// TIA Portal V17 export
// export: Created 2024-09-03T21:54:49.3245379Z, ExportSetting WithDefaults, DisplayName Totally Integrated Automation Portal, DisplayVersion V17 Update 7, DisplayName TIA Portal Openness, DisplayVersion V17 Update 7, DisplayName TIA Portal Version Control Interface, DisplayVersion V17, DisplayName SINAMICS Startdrive Advanced, DisplayVersion V17 SP2, DisplayName SINAMICS Startdrive G110M, G120, G120C, G120D, G120P, G115D, DisplayVersion V17 SP2, DisplayName SINAMICS Startdrive G130, G150, S120, S150, SINAMICS MV, S210, DisplayVersion V17 SP2, DisplayName STEP 7 Professional, DisplayVersion V17 Update 7, DisplayName STEP 7 Safety, DisplayVersion V17 Update 6, DisplayName WinCC Advanced / Unified PC, DisplayVersion V17 Update 7
DATA_BLOCK "HydraulicMain_DB"   // DB55
VERSION : 0.1
// stored: AutoNumber true, DBAccessibleFromOPCUA true, DBAccessibleFromWebserver true, InstanceOfName HydraulicMain, InstanceOfType FB
"HydraulicMain"
   // VAR
   //    HydraulicCylinder_LeftCupforming { S7_SetPoint := 'True'} : "HydraulicCylinder";
   //    HydraulicCylinder_RightCupforming { S7_SetPoint := 'True'} : "HydraulicCylinder";
   //    VH1StatusOld { S7_SetPoint := 'True'} : "UDT_Cylinder";
   //    VH2StatusOld { S7_SetPoint := 'True'} : "UDT_Cylinder";
   //    VH3StatusOld { S7_SetPoint := 'True'} : "UDT_Cylinder";
   //    VH4StatusOld { S7_SetPoint := 'True'} : "UDT_Cylinder";
   //    FittingCycle_InstanceCupformingLeft { S7_SetPoint := 'True'} : "FittingCycle";
   //    FittingCycle_InstanceCupformingRight { S7_SetPoint := 'True'} : "FittingCycle";
   //    R_TRIG_Instance { S7_SetPoint := 'True'} : R_TRIG;
   //    R_TRIG_Instance_1 { S7_SetPoint := 'True'} : R_TRIG;
   //    R_TRIG_Instance_2 { S7_SetPoint := 'True'} : R_TRIG;
   //    R_TRIG_Instance_3 { S7_SetPoint := 'True'} : R_TRIG;
   //    HydraulicMotor_Instance { S7_SetPoint := 'True'} : "HydraulicMotor";
   //    dummyCylinderLeft { ExternalAccessible := 'False'; ExternalVisible := 'False'; ExternalWritable := 'False'} : "UDT_Cylinder";
   //    dummyCylinderRight { S7_SetPoint := 'True'} : "UDT_Cylinder";
   // END_VAR
BEGIN
   HydraulicCylinder_LeftCupforming.HydraulicActive := FALSE;
   HydraulicCylinder_LeftCupforming.BasicPositionMin := -5.0;
   HydraulicCylinder_LeftCupforming.BasicPositionMax := 10.0;
   HydraulicCylinder_LeftCupforming.MaxPosition := 105.0;
   HydraulicCylinder_LeftCupforming.ManualCommand := 0;
   HydraulicCylinder_LeftCupforming.CylinderNumber := 3;
   HydraulicCylinder_LeftCupforming.dataOld.Pressure := 0.0;
   HydraulicCylinder_LeftCupforming.dataOld.Flow := 0.0;
   HydraulicCylinder_LeftCupforming.dataOld.Position := 0.0;
   HydraulicCylinder_LeftCupforming.dataOld.StandstillPosition := 0.0;
   HydraulicCylinder_LeftCupforming.dataOld.PressureCmd := 0.0;
   HydraulicCylinder_LeftCupforming.dataOld.FlowCmd := 0.0;
   HydraulicCylinder_LeftCupforming.dataOld.PressureBack := 0.0;
   HydraulicCylinder_LeftCupforming.dataOld.FlowBack := 0.0;
   HydraulicCylinder_LeftCupforming.dataOld.HAxis := 0.0;
   HydraulicCylinder_LeftCupforming.dataOld.Force := 0.0;
   HydraulicCylinder_LeftCupforming.dataOld.Status.InWp := FALSE;
   HydraulicCylinder_LeftCupforming.dataOld.Status.InBp := TRUE;
   HydraulicCylinder_LeftCupforming.dataOld.Status.InFp := TRUE;
   HydraulicCylinder_LeftCupforming.dataOld.Status.ToWp := FALSE;
   HydraulicCylinder_LeftCupforming.dataOld.Status.ToBp := FALSE;
   HydraulicCylinder_LeftCupforming.dataOld.Status.ToFp := TRUE;
   HydraulicCylinder_LeftCupforming.noCollision := TRUE;
   HydraulicCylinder_LeftCupforming.IEC_Timer_0_Instance.PT := T#3S;
   HydraulicCylinder_LeftCupforming.IEC_Timer_0_Instance.IN := FALSE;
   HydraulicCylinder_LeftCupforming.R_TRIG_Instance.CLK := TRUE;
   HydraulicCylinder_LeftCupforming.R_TRIG_Instance.Q := FALSE;
   HydraulicCylinder_LeftCupforming.R_TRIG_Instance.Stat_Bit := TRUE;
   HydraulicCylinder_LeftCupforming.difference := -0.01085043;
   HydraulicCylinder_LeftCupforming.re := -0.1085043;
   HydraulicCylinder_LeftCupforming.IEC_Timer_0_Instance_1.PT := T#400MS;
   HydraulicCylinder_LeftCupforming.IEC_Timer_0_Instance_1.IN := TRUE;
   HydraulicCylinder_LeftCupforming.RampFunction_Instance.Output := 0.0;
   HydraulicCylinder_LeftCupforming.RampFunction_Instance.ErrorBits := 16#0000_0000;
   HydraulicCylinder_RightCupforming.HydraulicActive := FALSE;
   HydraulicCylinder_RightCupforming.BasicPositionMin := -5.0;
   HydraulicCylinder_RightCupforming.BasicPositionMax := 10.0;
   HydraulicCylinder_RightCupforming.MaxPosition := 105.0;
   HydraulicCylinder_RightCupforming.ManualCommand := 0;
   HydraulicCylinder_RightCupforming.CylinderNumber := 4;
   HydraulicCylinder_RightCupforming.dataOld.Pressure := 0.0;
   HydraulicCylinder_RightCupforming.dataOld.Flow := 0.0;
   HydraulicCylinder_RightCupforming.dataOld.Position := 0.0;
   HydraulicCylinder_RightCupforming.dataOld.StandstillPosition := 0.0;
   HydraulicCylinder_RightCupforming.dataOld.PressureCmd := 0.0;
   HydraulicCylinder_RightCupforming.dataOld.FlowCmd := 0.0;
   HydraulicCylinder_RightCupforming.dataOld.PressureBack := 0.0;
   HydraulicCylinder_RightCupforming.dataOld.FlowBack := 0.0;
   HydraulicCylinder_RightCupforming.dataOld.HAxis := 0.0;
   HydraulicCylinder_RightCupforming.dataOld.Force := 0.0;
   HydraulicCylinder_RightCupforming.dataOld.Status.InWp := FALSE;
   HydraulicCylinder_RightCupforming.dataOld.Status.InBp := TRUE;
   HydraulicCylinder_RightCupforming.dataOld.Status.InFp := TRUE;
   HydraulicCylinder_RightCupforming.dataOld.Status.ToWp := FALSE;
   HydraulicCylinder_RightCupforming.dataOld.Status.ToBp := FALSE;
   HydraulicCylinder_RightCupforming.dataOld.Status.ToFp := TRUE;
   HydraulicCylinder_RightCupforming.noCollision := TRUE;
   HydraulicCylinder_RightCupforming.IEC_Timer_0_Instance.PT := T#3S;
   HydraulicCylinder_RightCupforming.IEC_Timer_0_Instance.IN := FALSE;
   HydraulicCylinder_RightCupforming.R_TRIG_Instance.CLK := TRUE;
   HydraulicCylinder_RightCupforming.R_TRIG_Instance.Q := FALSE;
   HydraulicCylinder_RightCupforming.R_TRIG_Instance.Stat_Bit := TRUE;
   HydraulicCylinder_RightCupforming.difference := -0.006510258;
   HydraulicCylinder_RightCupforming.re := -0.06510258;
   HydraulicCylinder_RightCupforming.IEC_Timer_0_Instance_1.PT := T#400MS;
   HydraulicCylinder_RightCupforming.IEC_Timer_0_Instance_1.IN := TRUE;
   HydraulicCylinder_RightCupforming.RampFunction_Instance.Output := 0.0;
   HydraulicCylinder_RightCupforming.RampFunction_Instance.ErrorBits := 16#0000_0000;
   VH1StatusOld.InWp := FALSE;
   VH1StatusOld.InBp := FALSE;
   VH1StatusOld.InFp := FALSE;
   VH1StatusOld.ToWp := FALSE;
   VH1StatusOld.ToBp := FALSE;
   VH1StatusOld.ToFp := FALSE;
   VH2StatusOld.InWp := FALSE;
   VH2StatusOld.InBp := FALSE;
   VH2StatusOld.InFp := FALSE;
   VH2StatusOld.ToWp := FALSE;
   VH2StatusOld.ToBp := FALSE;
   VH2StatusOld.ToFp := FALSE;
   VH3StatusOld.InWp := FALSE;
   VH3StatusOld.InBp := FALSE;
   VH3StatusOld.InFp := FALSE;
   VH3StatusOld.ToWp := FALSE;
   VH3StatusOld.ToBp := FALSE;
   VH3StatusOld.ToFp := FALSE;
   VH4StatusOld.InWp := FALSE;
   VH4StatusOld.InBp := FALSE;
   VH4StatusOld.InFp := FALSE;
   VH4StatusOld.ToWp := FALSE;
   VH4StatusOld.ToBp := FALSE;
   VH4StatusOld.ToFp := FALSE;
   FittingCycle_InstanceCupformingLeft.parameters.DigiforceProgram := 1;
   FittingCycle_InstanceCupformingLeft.parameters.FinalSpeed := 25.0;
   FittingCycle_InstanceCupformingLeft.parameters.ApproachSpeed := 25.0;
   FittingCycle_InstanceCupformingLeft.parameters.FinalForce := 10.0;
   FittingCycle_InstanceCupformingLeft.parameters.ApproachForce := 10.0;
   FittingCycle_InstanceCupformingLeft.parameters.EndWayImmediate := 2.55;
   FittingCycle_InstanceCupformingLeft.parameters.EndWayWithTimeout := 3.0;
   FittingCycle_InstanceCupformingLeft.parameters.SwitchingWay := 20.0;
   FittingCycle_InstanceCupformingLeft.parameters.EndWayTimeout := T#300MS;
   FittingCycle_InstanceCupformingLeft.basicPosition := TRUE;
   FittingCycle_InstanceCupformingLeft.MaxPosition := 105.0;
   FittingCycle_InstanceCupformingLeft.endStopCylinderActive := TRUE;
   FittingCycle_InstanceCupformingLeft.shiftSupportToWork := FALSE;
   FittingCycle_InstanceCupformingLeft.cnt := 0;
   FittingCycle_InstanceCupformingLeft.R_TRIG_Instance.CLK := FALSE;
   FittingCycle_InstanceCupformingLeft.R_TRIG_Instance.Q := FALSE;
   FittingCycle_InstanceCupformingLeft.R_TRIG_Instance.Stat_Bit := FALSE;
   FittingCycle_InstanceCupformingLeft.H2Reached := TRUE;
   FittingCycle_InstanceCupformingLeft.IEC_Timer_timeout.PT := T#15S;
   FittingCycle_InstanceCupformingLeft.IEC_Timer_timeout.IN := FALSE;
   FittingCycle_InstanceCupformingLeft.DigiforceStarted := TRUE;
   FittingCycle_InstanceCupformingLeft.R_TRIG_Instance_1.CLK := FALSE;
   FittingCycle_InstanceCupformingLeft.R_TRIG_Instance_1.Q := FALSE;
   FittingCycle_InstanceCupformingLeft.R_TRIG_Instance_1.Stat_Bit := FALSE;
   FittingCycle_InstanceCupformingLeft.ton_WayWithTimeoutReached.PT := T#300MS;
   FittingCycle_InstanceCupformingLeft.ton_WayWithTimeoutReached.IN := FALSE;
   FittingCycle_InstanceCupformingRight.parameters.DigiforceProgram := 1;
   FittingCycle_InstanceCupformingRight.parameters.FinalSpeed := 25.0;
   FittingCycle_InstanceCupformingRight.parameters.ApproachSpeed := 25.0;
   FittingCycle_InstanceCupformingRight.parameters.FinalForce := 10.0;
   FittingCycle_InstanceCupformingRight.parameters.ApproachForce := 10.0;
   FittingCycle_InstanceCupformingRight.parameters.EndWayImmediate := 2.7;
   FittingCycle_InstanceCupformingRight.parameters.EndWayWithTimeout := 3.0;
   FittingCycle_InstanceCupformingRight.parameters.SwitchingWay := 20.0;
   FittingCycle_InstanceCupformingRight.parameters.EndWayTimeout := T#300MS;
   FittingCycle_InstanceCupformingRight.basicPosition := TRUE;
   FittingCycle_InstanceCupformingRight.MaxPosition := 105.0;
   FittingCycle_InstanceCupformingRight.endStopCylinderActive := TRUE;
   FittingCycle_InstanceCupformingRight.shiftSupportToWork := TRUE;
   FittingCycle_InstanceCupformingRight.cnt := 0;
   FittingCycle_InstanceCupformingRight.R_TRIG_Instance.CLK := FALSE;
   FittingCycle_InstanceCupformingRight.R_TRIG_Instance.Q := FALSE;
   FittingCycle_InstanceCupformingRight.R_TRIG_Instance.Stat_Bit := FALSE;
   FittingCycle_InstanceCupformingRight.H2Reached := TRUE;
   FittingCycle_InstanceCupformingRight.IEC_Timer_timeout.PT := T#15S;
   FittingCycle_InstanceCupformingRight.IEC_Timer_timeout.IN := FALSE;
   FittingCycle_InstanceCupformingRight.DigiforceStarted := TRUE;
   FittingCycle_InstanceCupformingRight.R_TRIG_Instance_1.CLK := FALSE;
   FittingCycle_InstanceCupformingRight.R_TRIG_Instance_1.Q := FALSE;
   FittingCycle_InstanceCupformingRight.R_TRIG_Instance_1.Stat_Bit := FALSE;
   FittingCycle_InstanceCupformingRight.ton_WayWithTimeoutReached.PT := T#300MS;
   FittingCycle_InstanceCupformingRight.ton_WayWithTimeoutReached.IN := FALSE;
   R_TRIG_Instance.CLK := FALSE;
   R_TRIG_Instance.Q := FALSE;
   R_TRIG_Instance.Stat_Bit := FALSE;
   R_TRIG_Instance_1.CLK := FALSE;
   R_TRIG_Instance_1.Q := FALSE;
   R_TRIG_Instance_1.Stat_Bit := FALSE;
   R_TRIG_Instance_2.CLK := FALSE;
   R_TRIG_Instance_2.Q := FALSE;
   R_TRIG_Instance_2.Stat_Bit := FALSE;
   R_TRIG_Instance_3.CLK := FALSE;
   R_TRIG_Instance_3.Q := FALSE;
   R_TRIG_Instance_3.Stat_Bit := FALSE;
   HydraulicMotor_Instance.cycleActiveCupforming := FALSE;
   HydraulicMotor_Instance.temp1nok := FALSE;
   HydraulicMotor_Instance.temp2nok := FALSE;
   HydraulicMotor_Instance.qKM20 := FALSE;
   HydraulicMotor_Instance.qMotor := FALSE;
   HydraulicMotor_Instance.qValveCupforming := FALSE;
   HydraulicMotor_Instance.R_TRIG_Instance.CLK := FALSE;
   HydraulicMotor_Instance.R_TRIG_Instance.Q := FALSE;
   HydraulicMotor_Instance.R_TRIG_Instance.Stat_Bit := FALSE;
   HydraulicMotor_Instance.cnt := 0;
   HydraulicMotor_Instance.IEC_Timer_0_Instance.PT := T#3S;
   HydraulicMotor_Instance.IEC_Timer_0_Instance.IN := FALSE;
   HydraulicMotor_Instance.F_TRIG_Instance.CLK := FALSE;
   HydraulicMotor_Instance.F_TRIG_Instance.Q := FALSE;
   HydraulicMotor_Instance.F_TRIG_Instance.Stat_Bit := FALSE;
   HydraulicMotor_Instance.IEC_Timer_0_Instance_1.PT := T#0MS;
   HydraulicMotor_Instance.IEC_Timer_0_Instance_1.IN := FALSE;
   dummyCylinderLeft.InWp := FALSE;
   dummyCylinderLeft.InBp := TRUE;
   dummyCylinderLeft.InFp := FALSE;
   dummyCylinderLeft.ToWp := FALSE;
   dummyCylinderLeft.ToBp := TRUE;
   dummyCylinderLeft.ToFp := FALSE;
   dummyCylinderRight.InWp := FALSE;
   dummyCylinderRight.InBp := TRUE;
   dummyCylinderRight.InFp := FALSE;
   dummyCylinderRight.ToWp := FALSE;
   dummyCylinderRight.ToBp := TRUE;
   dummyCylinderRight.ToFp := FALSE;
END_DATA_BLOCK
